DATA_BLOCK "DB_DualStarterCell"
{ S7_Optimized_Access := 'TRUE' }
VERSION : 0.1
NON_RETAIN
"FB_DualStarterCell"
BEGIN
END_DATA_BLOCK
